(* CoDeSys 2.3 export: ST_LP_FUNC_CFG.EXP *)

(* Data type *)
TYPE ST_LP_FUNC_CFG :
STRUCT
	SpdA_Min : REAL;
	SpdA_Max : REAL;
	SpdB_Min : REAL;
	SpdB_Max : REAL;

	Spd_Inc : REAL;
	Spd_Dec : REAL;

	A_Spd1 : BOOL;

	SF1_Limit : BOOL;
	SF2_Limit : BOOL;

	Cycle   : REAL; (*Seconds*)
	TimeMax : REAL; (*Seconds*)

(*	PP : BYTE;*)
END_STRUCT
END_TYPE
